TYPE ST_FireSystem_Events :
STRUCT
	CODetFault		:	BOOL;
	CODetWarning1	:	BOOL;
	CODetWarning2	: 	BOOL;
	CODetAlarm		:	BOOL;
	SmokeDetFault	:	BOOL;
	SmokeDetAlarm	:	BOOL;
	AlarmMuted		:	BOOL;
END_STRUCT
END_TYPE

(* stored: Version 1.1.0.1, ProductVersion 3.1.4026.18
   DUT ST_FireSystem_Events: Id {a47fa298-6191-40e3-abfb-fd566d2a024d} *)
